// Mitsubishi GX Works2 project: TEx02   PLC: Q02/Q02H

PROGRAM MAIN
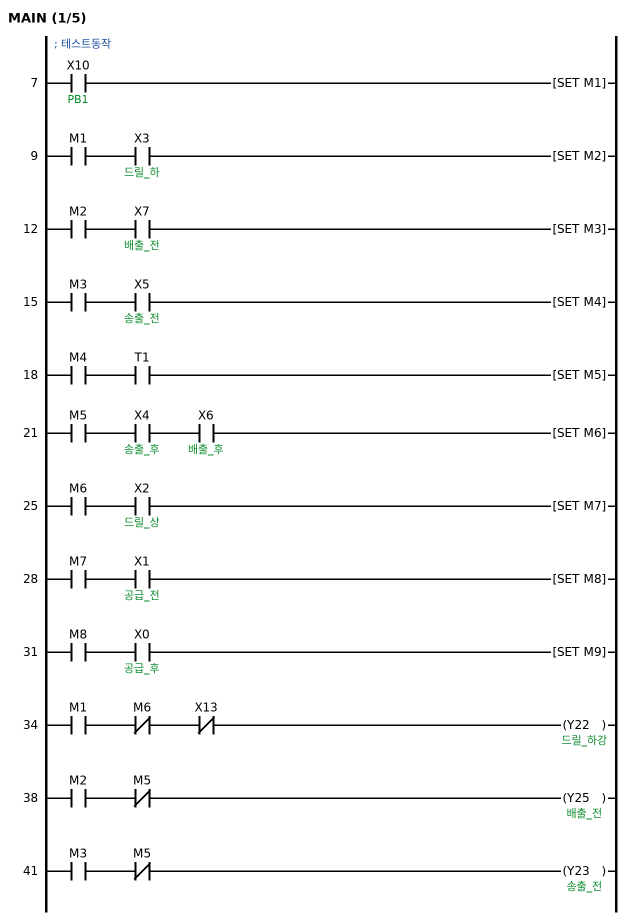
; 테스트동작
7     LD      X10  ; PB1
      SET     M1
9     LD      M1
      AND     X3  ; 드릴_하
      SET     M2
12    LD      M2
      AND     X7  ; 배출_전
      SET     M3
15    LD      M3
      AND     X5  ; 송출_전
      SET     M4
18    LD      M4
      AND     T1
      SET     M5
21    LD      M5
      AND     X4  ; 송출_후
      AND     X6  ; 배출_후
      SET     M6
25    LD      M6
      AND     X2  ; 드릴_상
      SET     M7
28    LD      M7
      AND     X1  ; 공급_전
      SET     M8
31    LD      M8
      AND     X0  ; 공급_후
      SET     M9
34    LD      M1
      ANI     M6
      ANI     X13
      OUT     Y22  ; 드릴_하강
38    LD      M2
      ANI     M5
      OUT     Y25  ; 배출_전
41    LD      M3
      ANI     M5
      OUT     Y23  ; 송출_전
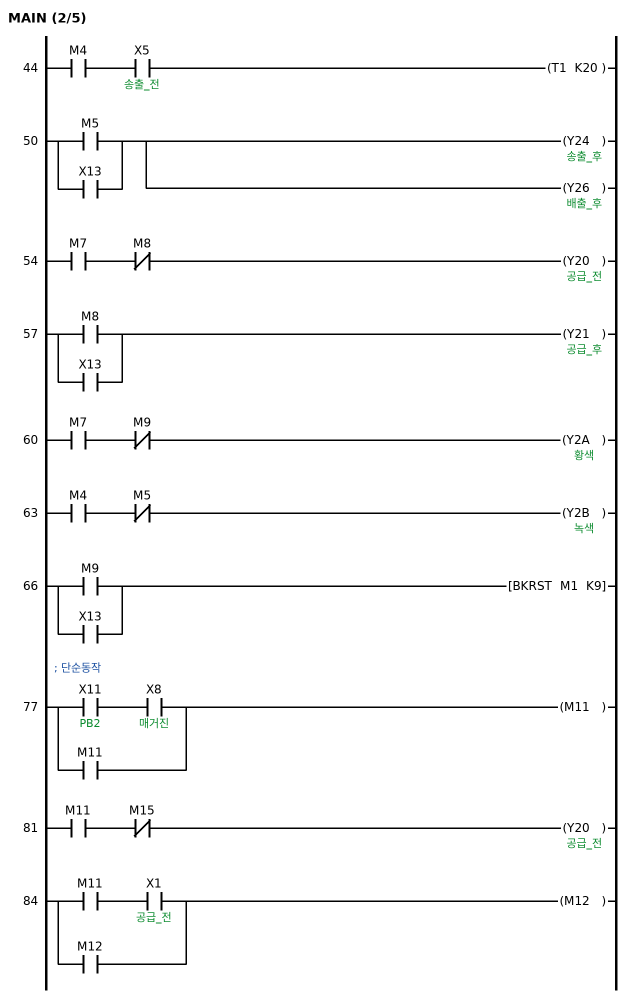
44    LD      M4
      AND     X5  ; 송출_전
      OUT     T1 K20
50    LD      M5
      OR      X13
      OUT     Y24  ; 송출_후
      OUT     Y26  ; 배출_후
54    LD      M7
      ANI     M8
      OUT     Y20  ; 공급_전
57    LD      M8
      OR      X13
      OUT     Y21  ; 공급_후
60    LD      M7
      ANI     M9
      OUT     Y2A  ; 황색
63    LD      M4
      ANI     M5
      OUT     Y2B  ; 녹색
66    LD      M9
      OR      X13
      BKRST   M1 K9
; 단순동작
77    LD      X11  ; PB2
      AND     X8  ; 매거진
      OR      M11
      OUT     M11
81    LD      M11
      ANI     M15
      OUT     Y20  ; 공급_전
84    LD      M11
      AND     X1  ; 공급_전
      OR      M12
      OUT     M12
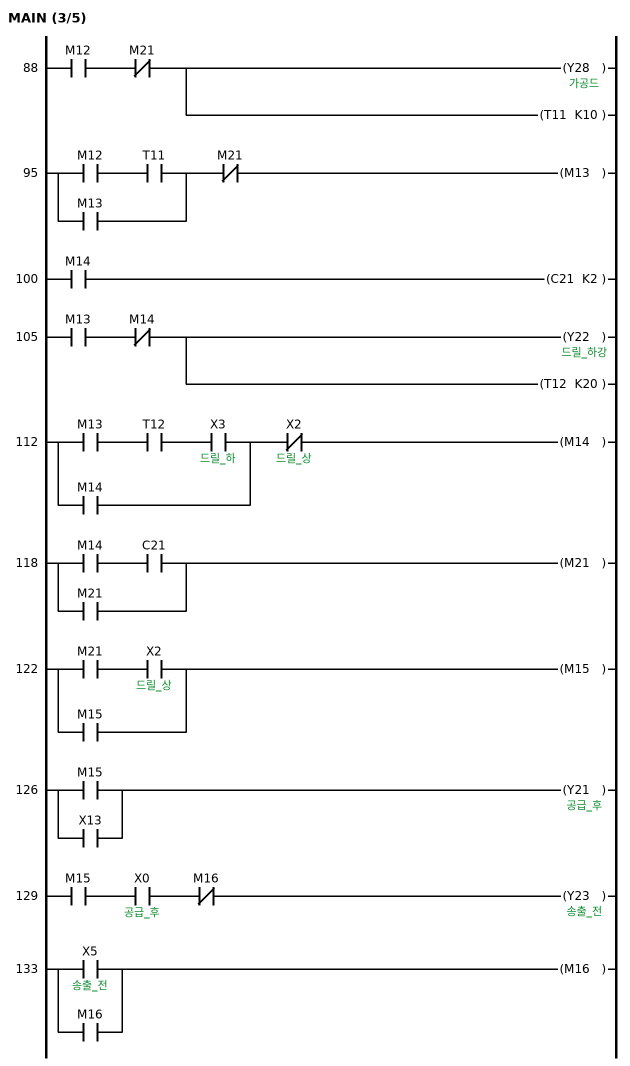
88    LD      M12
      ANI     M21
      OUT     Y28  ; 가공드
      OUT     T11 K10
95    LD      M12
      AND     T11
      OR      M13
      ANI     M21
      OUT     M13
100   LD      M14
      OUT     C21 K2
105   LD      M13
      ANI     M14
      OUT     Y22  ; 드릴_하강
      OUT     T12 K20
112   LD      M13
      AND     T12
      AND     X3  ; 드릴_하
      OR      M14
      ANI     X2  ; 드릴_상
      OUT     M14
118   LD      M14
      AND     C21
      OR      M21
      OUT     M21
122   LD      M21
      AND     X2  ; 드릴_상
      OR      M15
      OUT     M15
126   LD      M15
      OR      X13
      OUT     Y21  ; 공급_후
129   LD      M15
      AND     X0  ; 공급_후
      ANI     M16
      OUT     Y23  ; 송출_전
133   LD      X5  ; 송출_전
      OR      M16
      OUT     M16
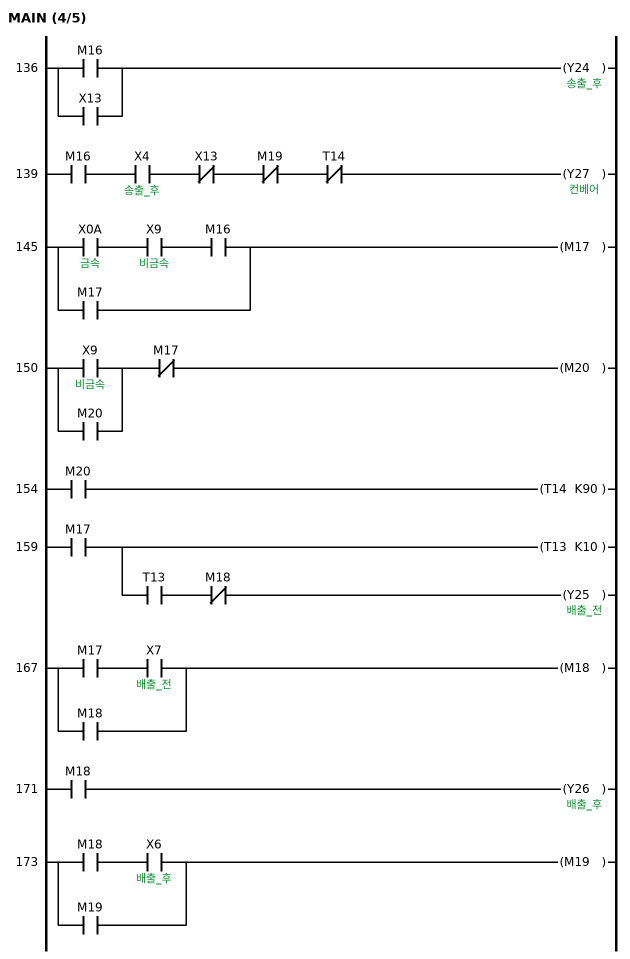
136   LD      M16
      OR      X13
      OUT     Y24  ; 송출_후
139   LD      M16
      AND     X4  ; 송출_후
      ANI     X13
      ANI     M19
      ANI     T14
      OUT     Y27  ; 컨베어
145   LD      X0A  ; 금속
      AND     X9  ; 비금속
      AND     M16
      OR      M17
      OUT     M17
150   LD      X9  ; 비금속
      OR      M20
      ANI     M17
      OUT     M20
154   LD      M20
      OUT     T14 K90
159   LD      M17
      OUT     T13 K10
      AND     T13
      ANI     M18
      OUT     Y25  ; 배출_전
167   LD      M17
      AND     X7  ; 배출_전
      OR      M18
      OUT     M18
171   LD      M18
      OUT     Y26  ; 배출_후
173   LD      M18
      AND     X6  ; 배출_후
      OR      M19
      OUT     M19
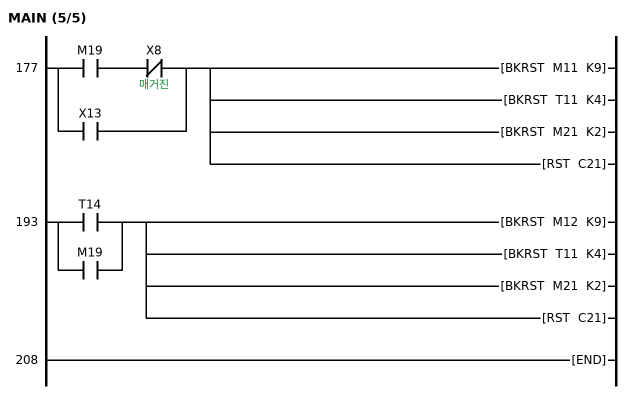
177   LD      M19
      ANI     X8  ; 매거진
      OR      X13
      BKRST   M11 K9
      BKRST   T11 K4
      BKRST   M21 K2
      RST     C21
193   LD      T14
      OR      M19
      BKRST   M12 K9
      BKRST   T11 K4
      BKRST   M21 K2
      RST     C21
208   END
END_PROGRAM

// device comments not shown above
X12  ; PB3
Y29  ; 적색
